// TIA Portal V18 export
DATA_BLOCK "DB_LHTTPParameters"   // DB6
{ S7_Optimized_Access := 'TRUE' }
// stored: MemoryReserve 100
   VAR
      hwID : HW_ANY;
      connID : CONN_OUC := 1;
      url : String := 'http://192.168.2.41:8885/data/v1/pipelines/getAccessLevel/value';   // 'http://192.168.2.41:8885/data/v1/pipelines/getAccessLevel/value'
      contentType : String := 'application/json';   // 'application/json'
      Head : String;
      HeaderData : Array[0..255] of Char;
      responseData : Array[0..1000] of Char;
   END_VAR
BEGIN
   HeaderData[0] := 'A';
   HeaderData[1] := 'u';
   HeaderData[2] := 't';
   HeaderData[3] := 'h';
   HeaderData[4] := 'o';
   HeaderData[5] := 'r';
   HeaderData[6] := 'i';
   HeaderData[7] := 'z';
   HeaderData[8] := 'a';
   HeaderData[9] := 't';
   HeaderData[10] := 'i';
   HeaderData[11] := 'o';
   HeaderData[12] := 'n';
   HeaderData[13] := ':';
   HeaderData[15] := 'B';
   HeaderData[16] := 'e';
   HeaderData[17] := 'a';
   HeaderData[18] := 'r';
   HeaderData[19] := 'e';
   HeaderData[20] := 'r';
   HeaderData[22] := 'm';
   HeaderData[23] := 'c';
   HeaderData[24] := 'p';
   HeaderData[25] := '2';
   HeaderData[26] := '.';
   HeaderData[27] := 'h';
   HeaderData[28] := 'E';
   HeaderData[29] := 'A';
   HeaderData[30] := 'n';
   HeaderData[31] := 'Q';
   HeaderData[32] := 'W';
   HeaderData[33] := '4';
   HeaderData[34] := 'o';
   HeaderData[35] := 's';
   HeaderData[36] := 'V';
   HeaderData[37] := '8';
   HeaderData[38] := 'l';
   HeaderData[39] := 'r';
   HeaderData[40] := 'Z';
   HeaderData[41] := 'T';
   HeaderData[42] := 'q';
   HeaderData[43] := 'w';
   HeaderData[44] := 'G';
   HeaderData[45] := '5';
   HeaderData[46] := 'f';
   HeaderData[47] := 'i';
   HeaderData[48] := 'v';
   HeaderData[49] := 'H';
   HeaderData[50] := 'Z';
   HeaderData[51] := 'n';
   HeaderData[52] := 'j';
   HeaderData[53] := '2';
   HeaderData[54] := 'C';
   HeaderData[55] := '7';
   HeaderData[56] := 'Q';
   HeaderData[57] := 'q';
   HeaderData[58] := 'l';
   HeaderData[59] := 'J';
   HeaderData[60] := 'w';
   HeaderData[61] := 'C';
   HeaderData[62] := 'K';
   HeaderData[63] := 'O';
   HeaderData[64] := 'i';
   HeaderData[65] := 'I';
   HeaderData[66] := '7';
   HeaderData[67] := 'R';
   HeaderData[68] := 'j';
   HeaderData[69] := 'c';
   HeaderData[70] := '=';
   HeaderData[71] := '$00';
END_DATA_BLOCK
